PROGRAM MAIN
VAR
END_VAR


	 
PRG_LivingRoom();

PRG_IoT_HMI_Connection();

END_PROGRAM

(* stored: Version 1.1.0.1, ProductVersion 3.1.4024.12
   POU MAIN: Id {fd0aff6f-dba4-40da-b5a8-b7bce76cd7be}, SpecialFunc None *)
